(* IEC 61131-3 sources: AXOpen/src/components.rexroth.tightening/ctrl/src/Axo_CS351_compact/TypesStructuresAndEnums, 15 files *)

(* ---- eAxo_CS351_compact_DataFormat.st ---- *)
NAMESPACE AXOpen.Components.Rexroth.Tightening
    TYPE PUBLIC
        eAxo_CS351_compact_DataFormat :
        (
            LittleEndian,
            BigEndian
        );
    END_TYPE
END_NAMESPACE

(* ---- eAxo_CS351_compacte_IoPointsSize.st ---- *)
NAMESPACE AXOpen.Components.Rexroth.Tightening
    TYPE PUBLIC
        eAxo_CS351_compacte_IoPointsSize :
        (
            _32bits_4bytes,
            _48bits_6bytes,
            _64bits_8bytes
        );
    END_TYPE
END_NAMESPACE

(* ---- Axo_CS351_compact_Component_Status.st ---- *)
NAMESPACE AXOpen.Components.Rexroth.Tightening
    {S7.extern=ReadWrite}
    {#ix-attr:[Container(Layout.Stack)]}
    CLASS PUBLIC Axo_CS351_compact_Component_Status EXTENDS AXOpen.Components.Abstractions.AxoComponent_Status
        VAR PUBLIC

        END_VAR
    END_CLASS
END_NAMESPACE

(* ---- Axo_CS351_compact_Config.st ---- *)
NAMESPACE AXOpen.Components.Rexroth.Tightening
    {S7.extern=ReadWrite}
    {#ix-attr:[Container(Layout.Stack)]}
    CLASS PUBLIC Axo_CS351_compact_Config
        VAR PUBLIC
            {#ix-set:AttributeName = "<#Info time#>"}
            InfoTime : LTIME := LT#5S;
            {#ix-set:AttributeName = "<#Error time#>"}
            ErrorTime : LTIME := LT#60S;
        END_VAR
    END_CLASS
END_NAMESPACE

(* ---- Axo_CS351_compact_Control.st ---- *)
NAMESPACE AXOpen.Components.Rexroth.Tightening
    {S7.extern=ReadWrite}
    {#ix-attr:[Container(Layout.Stack)]}
    CLASS PUBLIC Axo_CS351_compact_Control
        VAR PUBLIC
            // Signals : st_REX_CS351_ControlSignals;
            // Data : st_REX_CS351_ControlData;
        END_VAR
    END_CLASS
END_NAMESPACE

(* ---- Axo_CS351_compact_ControlData.st ---- *)
NAMESPACE AXOpen.Components.Rexroth.Tightening
    {S7.extern=ReadWrite}
    {#ix-attr:[Container(Layout.Stack)]}
    CLASS PUBLIC Axo_CS351_compact_ControlData
        VAR PUBLIC
            {#ix-set:AttributeName = "<#ID code#>"}
            IDcode : STRING;
        END_VAR
    END_CLASS
END_NAMESPACE

(* ---- Axo_CS351_compact_ControlSignals.st ---- *)
NAMESPACE AXOpen.Components.Rexroth.Tightening
    {S7.extern=ReadWrite}
    {#ix-attr:[Container(Layout.Stack)]}
    CLASS PUBLIC Axo_CS351_compact_ControlSignals
        VAR PUBLIC
            {#ix-set:AttributeName = "<#Program number#>"}
            ProgramNo : BYTE;
            {#ix-set:AttributeName = "<#Enable#>"}
            Enable : BOOL;
            {#ix-set:AttributeName = "<#Reset fault#>"}
            ResetFault : BOOL;
            {#ix-set:AttributeName = "<#Start clockwise#>"}
            StartClockwise : BOOL;
            {#ix-set:AttributeName = "<#Start counter clockwise#>"}
            StartCounterClockwise : BOOL;
            {#ix-set:AttributeName = "<#Reset results#>"}
            ResetResults : BOOL;
            {#ix-set:AttributeName = "<#Nok acknowledge#>"}
            NokAck : BOOL;
            {#ix-set:AttributeName = "<#User In 1#>"}
            UsrIn1 : BOOL;
            {#ix-set:AttributeName = "<#User In 2#>"}
            UsrIn2 : BOOL;
            {#ix-set:AttributeName = "<#ErgoSpin LED Green#>"}
            ES_LED_Green : BOOL;
            {#ix-set:AttributeName = "<#ErgoSpin LED Yellow#>"}
            ES_LED_Yellow : BOOL;
            {#ix-set:AttributeName = "<#ErgoSpin LED Red#>"}
            ES_LED_Red : BOOL;
            {#ix-set:AttributeName = "<#Active enable#>"}
            ActiveEnable : BOOL;
            {#ix-set:AttributeName = "<#Counter clockwise lock#>"}
            CcwLock : BOOL;
            {#ix-set:AttributeName = "<#Clockwise lock#>"}
            CwLock : BOOL;
            {#ix-set:AttributeName = "<#Clockwise AND#>"}
            CwAnd : BOOL;
            {#ix-set:AttributeName = "<#Counter clockwise AND#>"}
            CcwAND : BOOL;
        END_VAR
    END_CLASS
END_NAMESPACE

(* ---- Axo_CS351_compact_DATA.st ---- *)
NAMESPACE AXOpen.Components.Rexroth.Tightening
    {S7.extern=ReadWrite}
    {#ix-attr:[Container(Layout.Stack)]}
    CLASS PUBLIC Axo_CS351_compact_DATA
        VAR PUBLIC
            // Inputs : st_REX_CS351_Inputs;
            // Outputs : st_REX_CS351_Outputs;
        END_VAR
    END_CLASS
END_NAMESPACE

(* ---- Axo_CS351_compact_IDcode.st ---- *)
NAMESPACE AXOpen.Components.Rexroth.Tightening
    {S7.extern=ReadWrite}
    CLASS PUBLIC Axo_CS351_compact_IDcode EXTENDS AXOpen.Core.AxoByteArray
        VAR PUBLIC
            Data : ARRAY [0..15] OF BYTE;
        END_VAR
    END_CLASS
END_NAMESPACE

(* ---- Axo_CS351_compact_In.st ---- *)
NAMESPACE AXOpen.Components.Rexroth.Tightening
    {S7.extern=ReadWrite}
    {#ix-attr:[Container(Layout.Wrap)]}
    CLASS PUBLIC Axo_CS351_compact_In
        VAR PUBLIC
            {#ix-set:AttributeName = "<#Program number ack.#>"}
            ProgramNoAck : BYTE;
            {#ix-set:AttributeName = "<#Ready#>"}
            Ready : BOOL;
            {#ix-set:AttributeName = "<#No fault#>"}
            NoFault : BOOL;
            {#ix-set:AttributeName = "<#In Cycle#>"}
            InCycle : BOOL;
            {#ix-set:AttributeName = "<#In Cycle counter clockwise#>"}
            InCycleCcw : BOOL;
            {#ix-set:AttributeName = "<#Cycle complete#>"}
            CycleComplete : BOOL;
            {#ix-set:AttributeName = "<#OK#>"}
            OK : BOOL;
            {#ix-set:AttributeName = "<#NOK#>"}
            NOK : BOOL;
            {#ix-set:AttributeName = "<#Tool button#>"}
            ToolButton : BOOL;
            {#ix-set:AttributeName = "<#Counter clockwise select#>"}
            CcwSelect : BOOL;
            {#ix-set:AttributeName = "<#Start button ErgoSpin#>"}
            StartButton : BOOL;
            {#ix-set:AttributeName = "<#Triger Out#>"}
            TrigOut : BOOL;
            {#ix-set:AttributeName = "<#Torque too high#>"}
            TorqueHigh : BOOL;
            {#ix-set:AttributeName = "<#Torque too low#>"}
            TorqueLow : BOOL;
            {#ix-set:AttributeName = "<#Angle too high#>"}
            AngleHigh : BOOL;
            {#ix-set:AttributeName = "<#Angle too low#>"}
            AngleLow : BOOL;
            {#ix-set:AttributeName = "<#Counter clockwise lock acknowledge#>"}
            CcwLockAck : BOOL;
            {#ix-set:AttributeName = "<#Enable acknowledge#>"}
            EnableAck : BOOL;
            {#ix-set:AttributeName = "<#Active enable acknowledge#>"}
            ActiveEnableAck : BOOL;
            {#ix-set:AttributeName = "<#Clockwise lock acknowledge#>"}
            CwLockAck : BOOL;
            {#ix-set:AttributeName = "<#Clockwise acknowledge#>"}
            CwAck : BOOL;
            {#ix-set:AttributeName = "<#Counter clockwise acknowledge#>"}
            CcwAck : BOOL;
            {#ix-set:AttributeName = "<#ErgoSpin LED Green acknowledge#>"}
            ES_LED_GreenAck : BOOL;
            {#ix-set:AttributeName = "<#ErgoSpin LED Yellow acknowledge#>"}
            ES_LED_YellowAck : BOOL;
            {#ix-set:AttributeName = "<#ErgoSpin LED Red acknowledge#>"}
            ES_LED_RedAck : BOOL;
            {#ix-set:AttributeName = "<#Result#>"}
            Result : BYTE;
            // {#ix-set:AttributeName = "<#ID code#>"}
            IDcode : ARRAY[0..63] OF BYTE;
            {#ix-set:AttributeName = "<#Cycle counter#>"}
            CnoSE : UDINT;
            {#ix-set:AttributeName = "<#Program number#>"}
            ProgramNo : BYTE;
            {#ix-set:AttributeName = "<#Torque min#>"}
            TorqueMin : REAL;
            {#ix-set:AttributeName = "<#Torque#>"}
            Torque : REAL;
            {#ix-set:AttributeName = "<#Torque max#>"}
            TorqueMax : REAL;
            {#ix-set:AttributeName = "<#Angle min#>"}
            AngleMin : REAL;
            {#ix-set:AttributeName = "<#Angle#>"}
            Angle : REAL;
            {#ix-set:AttributeName = "<#Angle max#>"}
            AngleMax : REAL;
            {#ix-set:AttributeName = "<#Error code#>"}
            ErrorCode : INT;
            {#ix-set:AttributeName = "<#Error class#>"}
            ErrorClass : INT;
        END_VAR
    END_CLASS
END_NAMESPACE

(* ---- Axo_CS351_compact_Out.st ---- *)
NAMESPACE AXOpen.Components.Rexroth.Tightening
    {S7.extern=ReadWrite}
    {#ix-attr:[Container(Layout.Wrap)]}
    CLASS PUBLIC Axo_CS351_compact_Out
        VAR PUBLIC
            {#ix-set:AttributeName = "<#Control#>"}
            {#ix-attr:[ReadOnly()]}
            {#ix-set:AttributeName = "<#Program number#>"}
            ProgramNo : BYTE;
            {#ix-set:AttributeName = "<#Enable#>"}
            Enable : BOOL;
            {#ix-set:AttributeName = "<#Reset fault#>"}
            ResetFault : BOOL;
            {#ix-set:AttributeName = "<#Start clockwise#>"}
            StartClockwise : BOOL;
            {#ix-set:AttributeName = "<#Start counter clockwise#>"}
            StartCounterClockwise : BOOL;
            {#ix-set:AttributeName = "<#Reset results#>"}
            ResetResults : BOOL;
            {#ix-set:AttributeName = "<#Nok acknowledge#>"}
            NokAck : BOOL;
            {#ix-set:AttributeName = "<#User In 1#>"}
            UsrIn1 : BOOL;
            {#ix-set:AttributeName = "<#User In 2#>"}
            UsrIn2 : BOOL;
            {#ix-set:AttributeName = "<#ErgoSpin LED Green#>"}
            ES_LED_Green : BOOL;
            {#ix-set:AttributeName = "<#ErgoSpin LED Yellow#>"}
            ES_LED_Yellow : BOOL;
            {#ix-set:AttributeName = "<#ErgoSpin LED Red#>"}
            ES_LED_Red : BOOL;
            {#ix-set:AttributeName = "<#Active enable#>"}
            ActiveEnable : BOOL;
            {#ix-set:AttributeName = "<#Counter clockwise lock#>"}
            CcwLock : BOOL;
            {#ix-set:AttributeName = "<#Clockwise lock#>"}
            CwLock : BOOL;
            {#ix-set:AttributeName = "<#Clockwise AND#>"}
            CwAnd : BOOL;
            {#ix-set:AttributeName = "<#Counter clockwise AND#>"}
            CcwAND : BOOL;
            {#ix-set:AttributeName = "<#ID code#>"}
            IDcode : ARRAY[0..63] OF BYTE;
        END_VAR
    END_CLASS
END_NAMESPACE

(* ---- Axo_CS351_compact_QualityCode.st ---- *)
NAMESPACE AXOpen.Components.Rexroth.Tightening
    {S7.extern=ReadWrite}
    CLASS PUBLIC Axo_CS351_compact_QualityCode EXTENDS AXOpen.Core.AxoByteArray
        VAR PUBLIC
            Data : ARRAY [0..4] OF BYTE;
        END_VAR
    END_CLASS
END_NAMESPACE

(* ---- Axo_CS351_compact_Results.st ---- *)
NAMESPACE AXOpen.Components.Rexroth.Tightening
    {S7.extern=ReadWrite}
    {#ix-attr:[Container(Layout.Wrap)]}
    CLASS PUBLIC Axo_CS351_compact_Results
        VAR PUBLIC
            {#ix-set:AttributeName = "<#Result#>"}
            Result : BYTE;
            // {#ix-set:AttributeName = "<#ID code#>"}
            // {#ix-set:DisplayFormat = "string"}
            IDcode : ARRAY[0..63] OF BYTE;
            {#ix-set:AttributeName = "<#Cycle counter#>"}
            CnoSE : UDINT;
            {#ix-set:AttributeName = "<#Program number#>"}
            ProgramNo : BYTE;
            {#ix-set:AttributeName = "<#Torque min#>"}
            TorqueMin : REAL;
            {#ix-set:AttributeName = "<#Torque#>"}
            Torque : REAL;
            {#ix-set:AttributeName = "<#Torque max#>"}
            TorqueMax : REAL;
            {#ix-set:AttributeName = "<#Angle min#>"}
            AngleMin : REAL;
            {#ix-set:AttributeName = "<#Angle#>"}
            Angle : REAL;
            {#ix-set:AttributeName = "<#Angle max#>"}
            AngleMax : REAL;
            {#ix-set:AttributeName = "<#Error code#>"}
            ErrorCode : WORD;
            {#ix-set:AttributeName = "<#Error class#>"}
            ErrorClass : WORD;
        END_VAR
    END_CLASS
END_NAMESPACE

(* ---- Axo_CS351_compact_Status.st ---- *)
NAMESPACE AXOpen.Components.Rexroth.Tightening
    {S7.extern=ReadWrite}
    {#ix-attr:[Container(Layout.Stack)]}
    CLASS PUBLIC Axo_CS351_compact_Status
        VAR PUBLIC
            // Signals : st_REX_CS351_StateSignals;
            // Data : st_REX_CS351_ResultData;
        END_VAR
    END_CLASS
END_NAMESPACE

(* ---- Axo_CS351_HWIDs.st ---- *)
NAMESPACE AXOpen.Components.Rexroth.Tightening
    {S7.extern=ReadWrite}
     CLASS Axo_CS351_HWIDs
       VAR PUBLIC
          {#ix-set:AttributeName = "<#Hardware ID of the device#>"}
          HW_Device              : UINT;
          {#ix-set:AttributeName = "<#Hardware ID 'Slot 1' module#>"}
          HwID_Slot_1         :   UINT;
          {#ix-set:AttributeName = "<#Hardware ID 'Slot 2' module#>"}
          HwID_Slot_2         :   UINT;
          {#ix-set:AttributeName = "<#Hardware ID 'Slot 3' module#>"}
          HwID_Slot_3         :   UINT;
          {#ix-set:AttributeName = "<#Hardware ID 'Slot 4' module#>"}
          HwID_Slot_4         :   UINT;
          {#ix-set:AttributeName = "<#Hardware ID 'Slot 5' module#>"}
          HwID_Slot_5         :   UINT;
          {#ix-set:AttributeName = "<#Hardware ID 'Slot 6' module#>"}
          HwID_Slot_6         :   UINT;
          {#ix-set:AttributeName = "<#Hardware ID 'Slot 7' module#>"}
          HwID_Slot_7         :   UINT;
          {#ix-set:AttributeName = "<#Hardware ID 'Slot 8' module#>"}
          HwID_Slot_8         :   UINT;
          {#ix-set:AttributeName = "<#Hardware ID 'Slot 9' module#>"}
          HwID_Slot_9         :   UINT;
          {#ix-set:AttributeName = "<#Hardware ID 'Slot 10' module#>"}
          HwID_Slot_10        :   UINT;
          {#ix-set:AttributeName = "<#Hardware ID 'Slot 11' module#>"}
          HwID_Slot_11        :   UINT;
          {#ix-set:AttributeName = "<#Hardware ID 'Slot 12' module#>"}
          HwID_Slot_12        :   UINT;
          {#ix-set:AttributeName = "<#Hardware ID 'Slot 13' module#>"}
          HwID_Slot_13        :   UINT;
          {#ix-set:AttributeName = "<#Hardware ID 'Slot 14' module#>"}
          HwID_Slot_14        :   UINT;
          {#ix-set:AttributeName = "<#Hardware ID 'Slot 15' module#>"}
          HwID_Slot_15        :   UINT;
          {#ix-set:AttributeName = "<#Hardware ID 'Slot 16' module#>"}
          HwID_Slot_16        :   UINT;
          {#ix-set:AttributeName = "<#Hardware ID 'Slot 17' module#>"}
          HwID_Slot_17        :   UINT;
          {#ix-set:AttributeName = "<#Hardware ID 'Slot 18' module#>"}
          HwID_Slot_18        :   UINT;
          {#ix-set:AttributeName = "<#Hardware ID 'Slot 19' module#>"}
          HwID_Slot_19        :   UINT;
          {#ix-set:AttributeName = "<#Hardware ID 'Slot 20' module#>"}
          HwID_Slot_20        :   UINT;
          {#ix-set:AttributeName = "<#Hardware ID 'Slot 21' module#>"}
          HwID_Slot_21        :   UINT;
          {#ix-set:AttributeName = "<#Hardware ID 'Slot 22' module#>"}
          HwID_Slot_22        :   UINT;
          {#ix-set:AttributeName = "<#Hardware ID 'Slot 23' module#>"}
          HwID_Slot_23        :   UINT;
          {#ix-set:AttributeName = "<#Hardware ID 'Slot 24' module#>"}
          HwID_Slot_24        :   UINT;
          {#ix-set:AttributeName = "<#Hardware ID 'Slot 25' module#>"}
          HwID_Slot_25        :   UINT;
          {#ix-set:AttributeName = "<#Hardware ID 'Slot 26' module#>"}
          HwID_Slot_26        :   UINT;
       END_VAR
    END_CLASS
 END_NAMESPACE
